(* Logix 5000 project; controller Safety vendor 1 type 14 code 86 rev 19.11; software revision 19.01; part 14 of 17 *)
(* tags used below, declared in another part *)
   FVNR_y778MTR080RC : CONFIGURABLE_ROUT;   // Shear Die Crank Motor FVNR Run Command
   FVR_y702MTR191_Flt : ALIAS FOR Flt_Starter.4;   // Rewind Pinch Roll Starter Fault ( 1= Fault)
   FVR_y702MTR191FC : CONFIGURABLE_ROUT;   // Rewind Pinch Roll FVR Fwd Command
   FVR_y702MTR191RC : CONFIGURABLE_ROUT;   // Rewind Pinch Roll FVR Rev Command
   FVR_y778MTR080_Flt : ALIAS FOR Flt_Starter.5;   // Shear Die Crank Starter Fault ( 1= Fault)
   FVR_y802MTR080_Flt : ALIAS FOR Flt_Starter.6;   // Stacker Side Guide Lift Starter Fault ( 1= Fault)
   FVR_y802MTR080FC : CONFIGURABLE_ROUT;   // Stacker Side Guide Lift FVR Fwd Command
   FVR_y802MTR080RC : CONFIGURABLE_ROUT;   // Stacker Side Guide Lift FVR Rev Command
   FVR_y802MTR230_Flt : ALIAS FOR Flt_Starter.8;   // Scrap Horizontal Conveyor Starter Fault ( 1= Fault)
   FVR_y802MTR230FC : CONFIGURABLE_ROUT;   // Scrap Horizontal Conveyor FVR Fwd Command
   FVR_y802MTR230RC : CONFIGURABLE_ROUT;   // Scrap Horizontal Conveyor FVR Rev Command
   FVR_y802MTR231_Flt : ALIAS FOR Flt_Starter.7;   // Stacker Chain Conveyor Starter Fault ( 1= Fault)
   FVR_y802MTR231FC : CONFIGURABLE_ROUT;   // Stacker Chain Conveyor FVR Fwd Command
   FVR_y802MTR231RC : CONFIGURABLE_ROUT;   // Stacker Chain Conveyor FVR Rev Command
   Line_TotalMode : BOOL;   // Line TOTAL Mode ( 1= Total Mode) (0 = Coil to Coil)
   LineSts : UDT_SysStatus;
   OS11_S1_ModFlt : ALIAS FOR Flt_Modules[1].11;   // OS11 Point I/O Slot01 Module Fault (1 = Fault)
   OS13_S1_ModFlt : ALIAS FOR Flt_Modules[1].12;   // OS13 Point I/O Slot01 Module Fault (1 = Fault)
   OS14_S1_ModFlt : ALIAS FOR Flt_Modules[1].13;   // OS14 Point I/O Slot01 Module Fault (1 = Fault)
   OS15_S1_ModFlt : ALIAS FOR Flt_Modules[1].14;   // OS15 Point I/O Slot01 Module Fault (1 = Fault)
   OS16_S1_ModFlt : ALIAS FOR Flt_Modules[1].15;   // OS16 Point I/O Slot01 Module Fault (1 = Fault)
   OS1_S1_ModFlt : ALIAS FOR Flt_Modules[1].0;   // OS1 Point I/O Slot01 Module Fault (1 = Fault)
   OS2_S1_ModFlt : ALIAS FOR Flt_Modules[1].1;   // OS2 Point I/O Slot01 Module Fault (1 = Fault)
   OS3_S1_ModFlt : ALIAS FOR Flt_Modules[1].2;   // OS3 Point I/O Slot01 Module Fault (1 = Fault)
   OS4N_S1_ModFlt : ALIAS FOR Flt_Modules[1].3;   // OS4N Point I/O Slot01 Module Fault (1 = Fault)
   OS4N_S5_ModFlt : ALIAS FOR Flt_Modules[1].4;   // OS4N Point I/O Slot05 Module Fault (1 = Fault)
   OS4S_S1_ModFlt : ALIAS FOR Flt_Modules[1].5;   // OS4S Point I/O Slot01 Module Fault (1 = Fault)
   OS4S_S5_ModFlt : ALIAS FOR Flt_Modules[1].6;   // OS4S Point I/O Slot05 Module Fault (1 = Fault)
   OS5_S1_ModFlt : ALIAS FOR Flt_Modules[1].7;   // OS5 Point I/O Slot01 Module Fault (1 = Fault)
   OS6_S1_ModFlt : ALIAS FOR Flt_Modules[1].8;   // OS6 Point I/O Slot01 Module Fault (1 = Fault)
   OS8_S1_ModFlt : ALIAS FOR Flt_Modules[1].9;   // OS8 Point I/O Slot01 Module Fault (1 = Fault)
   OS9_S1_ModFlt : ALIAS FOR Flt_Modules[1].10;   // OS9 Point I/O Slot01 Module Fault (1 = Fault)
   RewPR_FVR_En : BOOL;   // Rewind Pinch Roll FVR Enable ( 1= Enable )
   RewPR_FVR_FltRst : BOOL;   // Rewind Pinch Roll Fault Reset ( 1= Reset Cmd )
   RewPR_FVR_FwdCmd : BOOL;   // Rewind Pinch Roll Forward Command ( 1= Run Fwd )
   RewPR_FVR_RevCmd : BOOL;   // Rewind Pinch Roll Reverse Command ( 1= Run Rev)
   ScHorCon_FVR_En : BOOL;   // Scrap Horizontal Conveyor FVR Enable ( 1= Enable )
   ScHorCon_FVR_FltRst : BOOL;   // Scrap Horizontal Conveyor Fault Reset ( 1= Reset Cmd )
   ScHorCon_FVR_FwdCmd : BOOL;   // Scrap Horizontal Conveyor Forward Command ( 1= Run Fwd )
   ScHorCon_FVR_RevCmd : BOOL;   // Scrap Horizontal Conveyor Reverse Command ( 1= Run Rev)
   SftyMap_Mach : DINT[5];   // SAFETY MAPPED From Machine Processor
   SftyMap_ShDie : DINT[5];   // SAFETY MAPPED From Shear Die Processor
   ShearSts : UDT_ShearStatus;
   SkChain_FVR_En : BOOL;   // Stacker Chain FVR Enable ( 1= Enable )
   SkChain_FVR_FltRst : BOOL;   // Stacker Chain Fault Reset ( 1= Reset Cmd )
   SkChain_FVR_FwdCmd : BOOL;   // Stacker Chain Forward Command ( 1= Run Fwd )
   SkChain_FVR_RevCmd : BOOL;   // Stacker Chain Reverse Command ( 1= Run Rev)
   SkSGLift_FVR_En : BOOL;   // Stacker Side Guide Lift FVR Enable ( 1= Enable )
   SkSGLift_FVR_FltRst : BOOL;   // Stacker Side Guide Lift Fault Reset ( 1= Reset Cmd )
   SkSGLift_FVR_FwdCmd : BOOL;   // Stacker Side Guide Lift Forward Command ( 1= Run Fwd )
   SkSGLift_FVR_RevCmd : BOOL;   // Stacker Side Guide Lift Reverse Command ( 1= Run Rev)
   SrDieCrnk_FVNR_En : BOOL;   // Shear Die Crank FVNR Enable ( 1= Enable )
   SrDieCrnk_FVNR_FltRst : BOOL;   // Shear Die Crank FVNR Enable ( 1= Enable )
   SrDieCrnk_FVNR_RunCmd : BOOL;   // Shear Die Crank Run Command ( 1= Run )
   x702MTR191FF : ALIAS FOR MCC1:1:I.Pt00Data;   // Rewind Pinch Roll Fwd Fdbk
   x702MTR191RF : ALIAS FOR MCC1:1:I.Pt01Data;   // Rewind Pinch Roll Rev Fdbk
   x778MTR080RF : ALIAS FOR MCC4:1:I.Pt00Data;   // Shear Crank Motor Run Fdbk
   x802MTR080FF : ALIAS FOR MCC5:1:I.Pt00Data;   // Stacker Side Guide Lift Fwd Fdbk/Up
   x802MTR080RF : ALIAS FOR MCC5:1:I.Pt01Data;   // Stacker Side Guide Lift Rev Fdbk/Down
   x802MTR230FF : ALIAS FOR MCC5:1:I.Pt02Data;   // Scrap Horizontal Conveyor Run Fwd Fdbk
   x802MTR230RF : ALIAS FOR MCC5:1:I.Pt03Data;   // Scrap Horizontal Conveyor Run Rev Fdbk
   x802MTR231FF : ALIAS FOR MCC5:1:I.Pt04Data;   // Stacker Chain Fwd Fdbk
   x802MTR231RF : ALIAS FOR MCC5:1:I.Pt05Data;   // Stacker Chain Rev Fdbk
   y702MTR191FC : ALIAS FOR MCC1:6:O.Pt00Data;   // Rewind Pinch Roll Fwd Cmd
   y702MTR191RC : ALIAS FOR MCC1:6:O.Pt01Data;   // Rewind Pinch Roll Rev Cmd
   y778MTR080RC : ALIAS FOR MCC4:4:O.Pt00Data;   // Shear Die Crank Run Cmd
   y802MTR080FC : ALIAS FOR MCC5:4:O.Pt04Data;   // Stacker Side Guide Lift Fwd Cmd/Up
   y802MTR080RC : ALIAS FOR MCC5:4:O.Pt05Data;   // Stacker Side Guide Lift Rev Cmd/Down
   y802MTR230FC : ALIAS FOR MCC5:4:O.Pt06Data;   // Scrap Horizontal Conveyor Fwd Cmd
   y802MTR230RC : ALIAS FOR MCC5:4:O.Pt07Data;   // Scrap Horizontal Conveyor Rev Cmd
   y802MTR231FC : ALIAS FOR MCC5:5:O.Pt00Data;   // Stacker Chain Fwd Cmd
   y802MTR231RC : ALIAS FOR MCC5:5:O.Pt01Data;   // Stacker Chain Rev Cmd
(* Starters, continued *)

ROUTINE A05_RewPR_FVR   (* ladder *)
// Rewind Pinch Roll
// FVR Starter
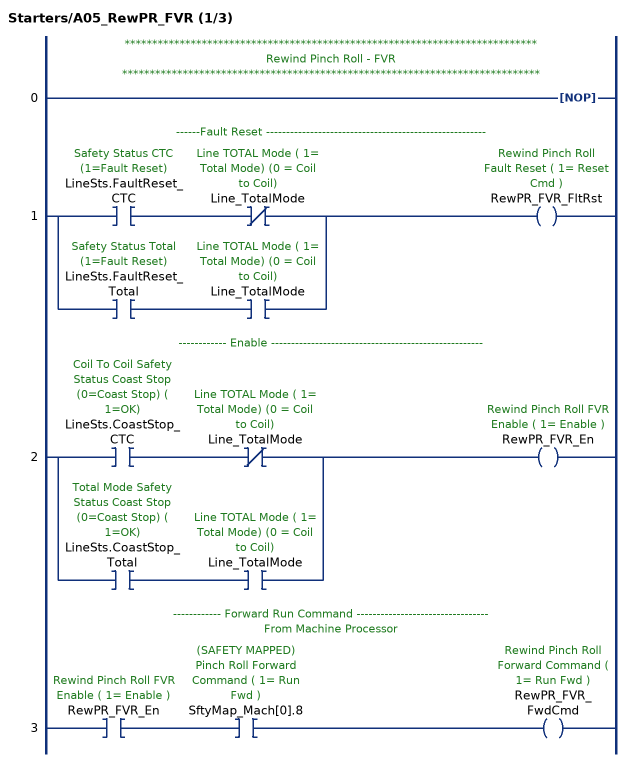
   // ***************************************************************************
   // Rewind Pinch Roll - FVR
   // ****************************************************************************
   0: NOP();
   // ------Fault Reset -------------------------------------------------------
   1: [XIC(LineSts.FaultReset_CTC) XIO(Line_TotalMode) ,XIC(LineSts.FaultReset_Total) XIC(Line_TotalMode) ]OTE(RewPR_FVR_FltRst);
   // ------------ Enable -----------------------------------------------------
   2: [XIC(LineSts.CoastStop_CTC) XIO(Line_TotalMode) ,XIC(LineSts.CoastStop_Total) XIC(Line_TotalMode) ]OTE(RewPR_FVR_En);
   // ------------ Forward Run Command ---------------------------------
   // From Machine Processor
   3: XIC(RewPR_FVR_En)XIC(SftyMap_Mach[0].8)OTE(RewPR_FVR_FwdCmd);
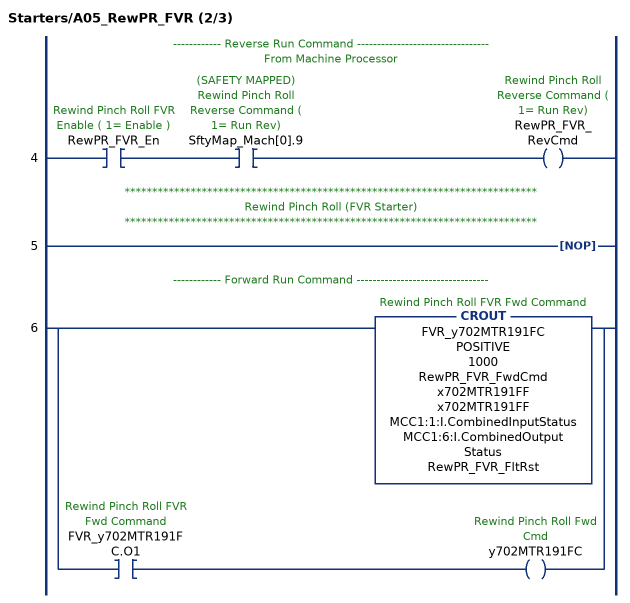
   // ------------ Reverse Run Command ---------------------------------
   // From Machine Processor
   4: XIC(RewPR_FVR_En)XIC(SftyMap_Mach[0].9)OTE(RewPR_FVR_RevCmd);
   // ***************************************************************************
   // Rewind Pinch Roll (FVR Starter)
   // ***************************************************************************
   5: NOP();
   // ------------ Forward Run Command ---------------------------------
   6: [CROUT(FVR_y702MTR191FC,POSITIVE,1000,RewPR_FVR_FwdCmd,x702MTR191FF,x702MTR191FF,MCC1:1:I.CombinedInputStatus,MCC1:6:I.CombinedOutputStatus,RewPR_FVR_FltRst) ,XIC(FVR_y702MTR191FC.O1) OTE(y702MTR191FC) ];
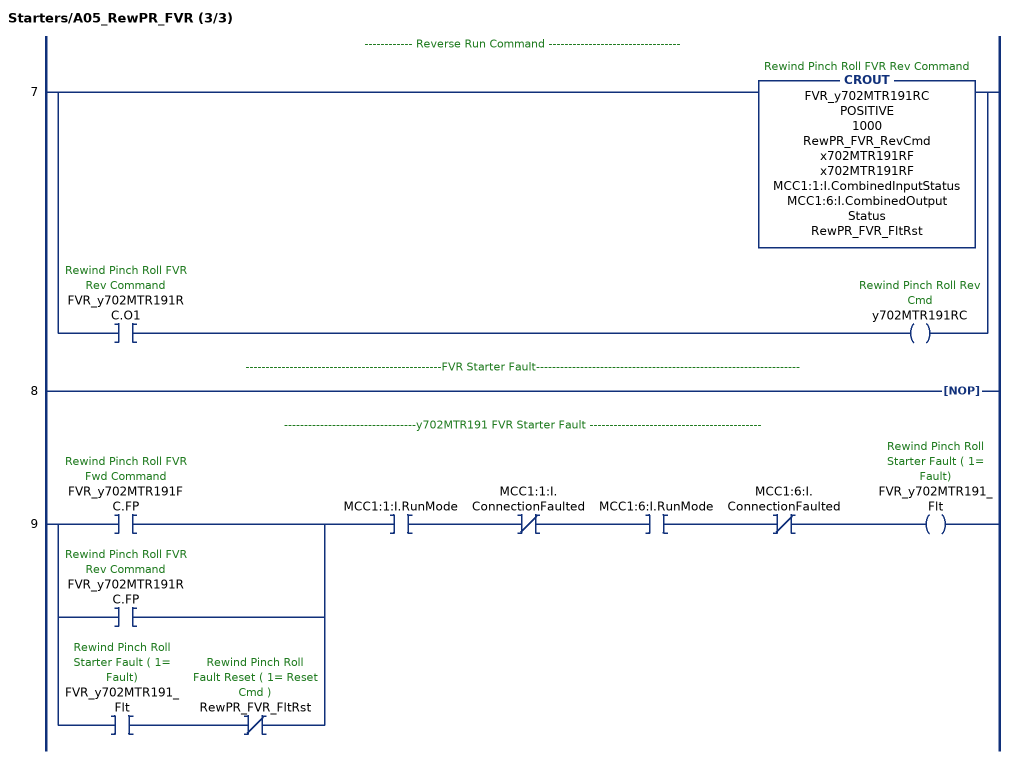
   // ------------ Reverse Run Command ---------------------------------
   7: [CROUT(FVR_y702MTR191RC,POSITIVE,1000,RewPR_FVR_RevCmd,x702MTR191RF,x702MTR191RF,MCC1:1:I.CombinedInputStatus,MCC1:6:I.CombinedOutputStatus,RewPR_FVR_FltRst) ,XIC(FVR_y702MTR191RC.O1) OTE(y702MTR191RC) ];
   // -------------------------------------------------FVR Starter Fault------------------------------------------------------------------
   8: NOP();
   // ---------------------------------y702MTR191 FVR Starter Fault -------------------------------------------
   9: [[XIC(FVR_y702MTR191FC.FP) ,XIC(FVR_y702MTR191RC.FP) ] ,XIC(FVR_y702MTR191_Flt) XIO(RewPR_FVR_FltRst) ]XIC(MCC1:1:I.RunMode)XIO(MCC1:1:I.ConnectionFaulted)XIC(MCC1:6:I.RunMode)XIO(MCC1:6:I.ConnectionFaulted)OTE(FVR_y702MTR191_Flt);
END_ROUTINE

ROUTINE A06_SrDieCrnk_FVNR   (* ladder *)
// Shear Die Crank
// FVNR Starter
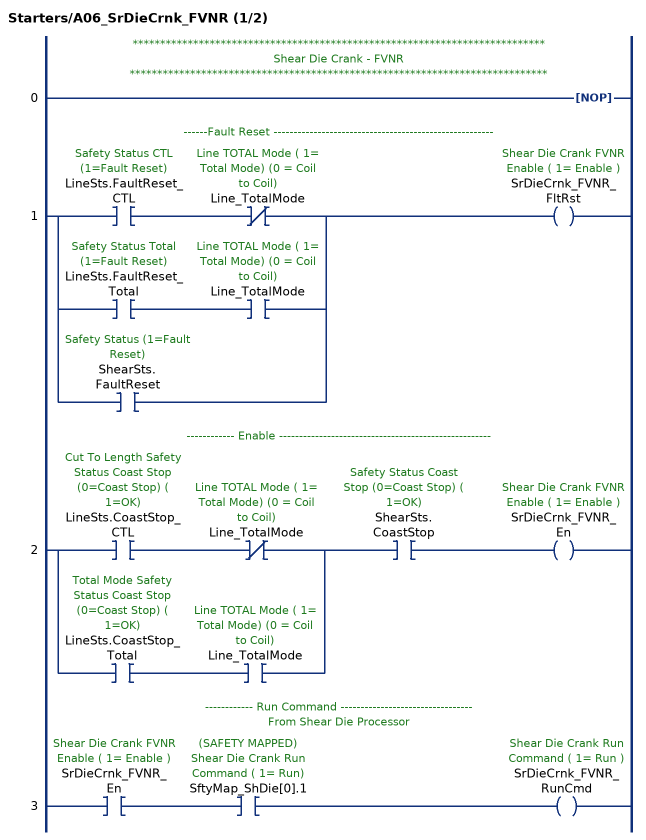
   // ***************************************************************************
   // Shear Die Crank - FVNR
   // ****************************************************************************
   0: NOP();
   // ------Fault Reset -------------------------------------------------------
   1: [XIC(LineSts.FaultReset_CTL) XIO(Line_TotalMode) ,XIC(LineSts.FaultReset_Total) XIC(Line_TotalMode) ,XIC(ShearSts.FaultReset) ]OTE(SrDieCrnk_FVNR_FltRst);
   // ------------ Enable -----------------------------------------------------
   2: [XIC(LineSts.CoastStop_CTL) XIO(Line_TotalMode) ,XIC(LineSts.CoastStop_Total) XIC(Line_TotalMode) ]XIC(ShearSts.CoastStop)OTE(SrDieCrnk_FVNR_En);
   // ------------ Run Command ---------------------------------
   // From Shear Die Processor
   3: XIC(SrDieCrnk_FVNR_En)XIC(SftyMap_ShDie[0].1)OTE(SrDieCrnk_FVNR_RunCmd);
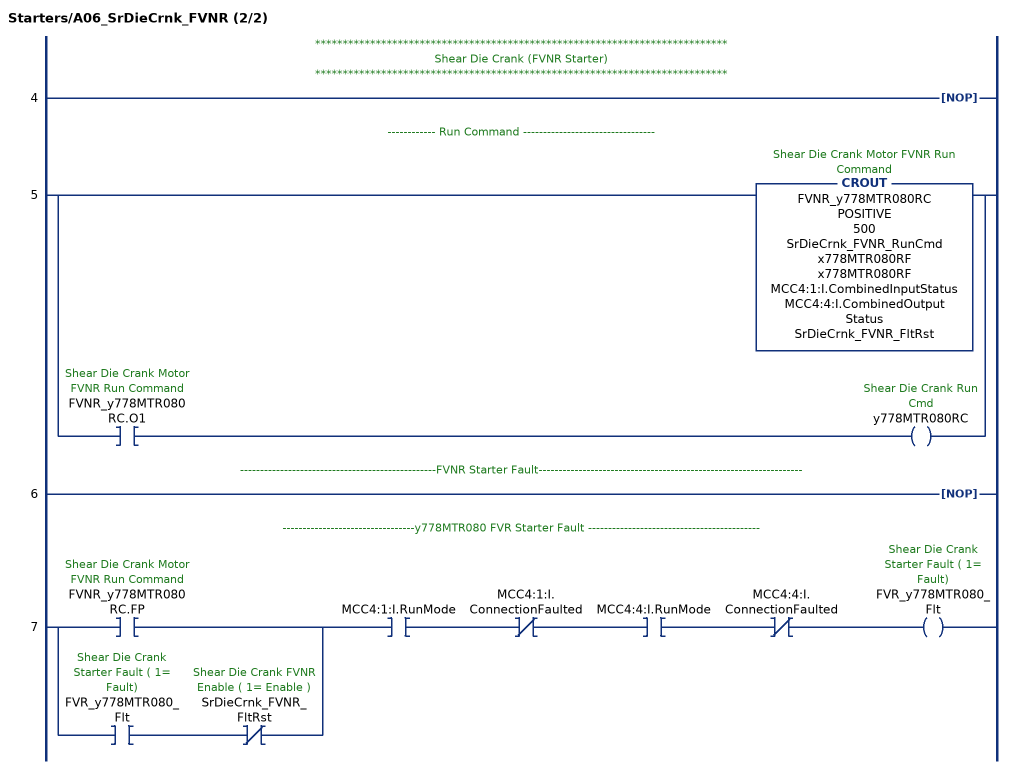
   // ***************************************************************************
   // Shear Die Crank (FVNR Starter)
   // ***************************************************************************
   4: NOP();
   // ------------ Run Command ---------------------------------
   5: [CROUT(FVNR_y778MTR080RC,POSITIVE,500,SrDieCrnk_FVNR_RunCmd,x778MTR080RF,x778MTR080RF,MCC4:1:I.CombinedInputStatus,MCC4:4:I.CombinedOutputStatus,SrDieCrnk_FVNR_FltRst) ,XIC(FVNR_y778MTR080RC.O1) OTE(y778MTR080RC) ];
   // -------------------------------------------------FVNR Starter Fault------------------------------------------------------------------
   6: NOP();
   // ---------------------------------y778MTR080 FVR Starter Fault -------------------------------------------
   7: [XIC(FVNR_y778MTR080RC.FP) ,XIC(FVR_y778MTR080_Flt) XIO(SrDieCrnk_FVNR_FltRst) ]XIC(MCC4:1:I.RunMode)XIO(MCC4:1:I.ConnectionFaulted)XIC(MCC4:4:I.RunMode)XIO(MCC4:4:I.ConnectionFaulted)OTE(FVR_y778MTR080_Flt);
END_ROUTINE

ROUTINE A07_SkSG_FVR   (* ladder *)
// Stacker Side Guide Lift
// FVR Starter
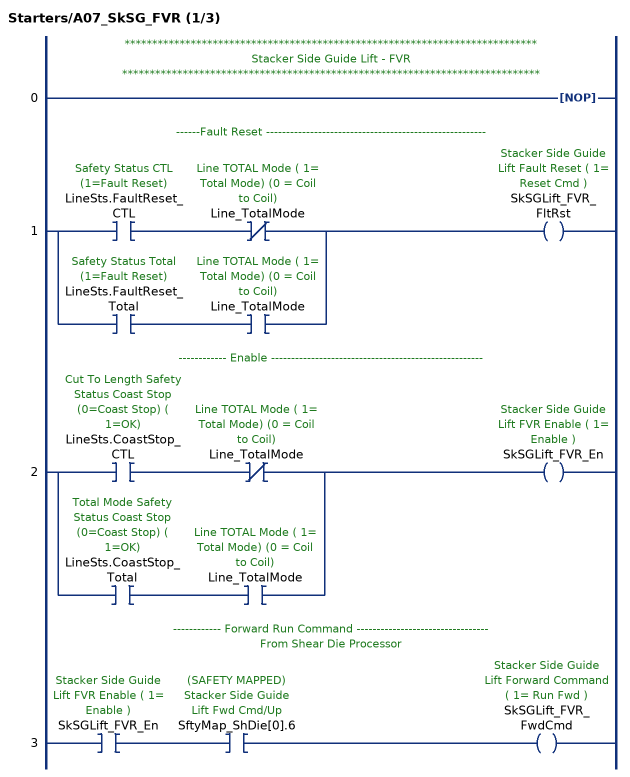
   // ***************************************************************************
   // Stacker Side Guide Lift - FVR
   // ****************************************************************************
   0: NOP();
   // ------Fault Reset -------------------------------------------------------
   1: [XIC(LineSts.FaultReset_CTL) XIO(Line_TotalMode) ,XIC(LineSts.FaultReset_Total) XIC(Line_TotalMode) ]OTE(SkSGLift_FVR_FltRst);
   // ------------ Enable -----------------------------------------------------
   2: [XIC(LineSts.CoastStop_CTL) XIO(Line_TotalMode) ,XIC(LineSts.CoastStop_Total) XIC(Line_TotalMode) ]OTE(SkSGLift_FVR_En);
   // ------------ Forward Run Command ---------------------------------
   // From Shear Die Processor
   3: XIC(SkSGLift_FVR_En)XIC(SftyMap_ShDie[0].6)OTE(SkSGLift_FVR_FwdCmd);
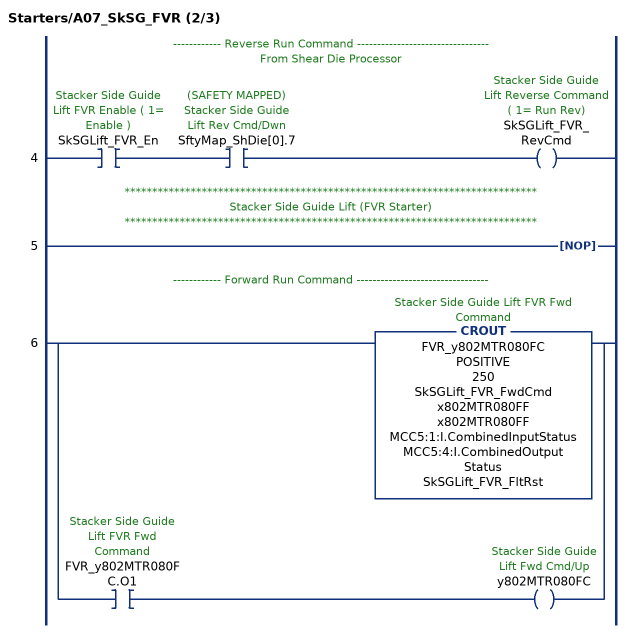
   // ------------ Reverse Run Command ---------------------------------
   // From Shear Die Processor
   4: XIC(SkSGLift_FVR_En)XIC(SftyMap_ShDie[0].7)OTE(SkSGLift_FVR_RevCmd);
   // ***************************************************************************
   // Stacker Side Guide Lift (FVR Starter)
   // ***************************************************************************
   5: NOP();
   // ------------ Forward Run Command ---------------------------------
   6: [CROUT(FVR_y802MTR080FC,POSITIVE,250,SkSGLift_FVR_FwdCmd,x802MTR080FF,x802MTR080FF,MCC5:1:I.CombinedInputStatus,MCC5:4:I.CombinedOutputStatus,SkSGLift_FVR_FltRst) ,XIC(FVR_y802MTR080FC.O1) OTE(y802MTR080FC) ];
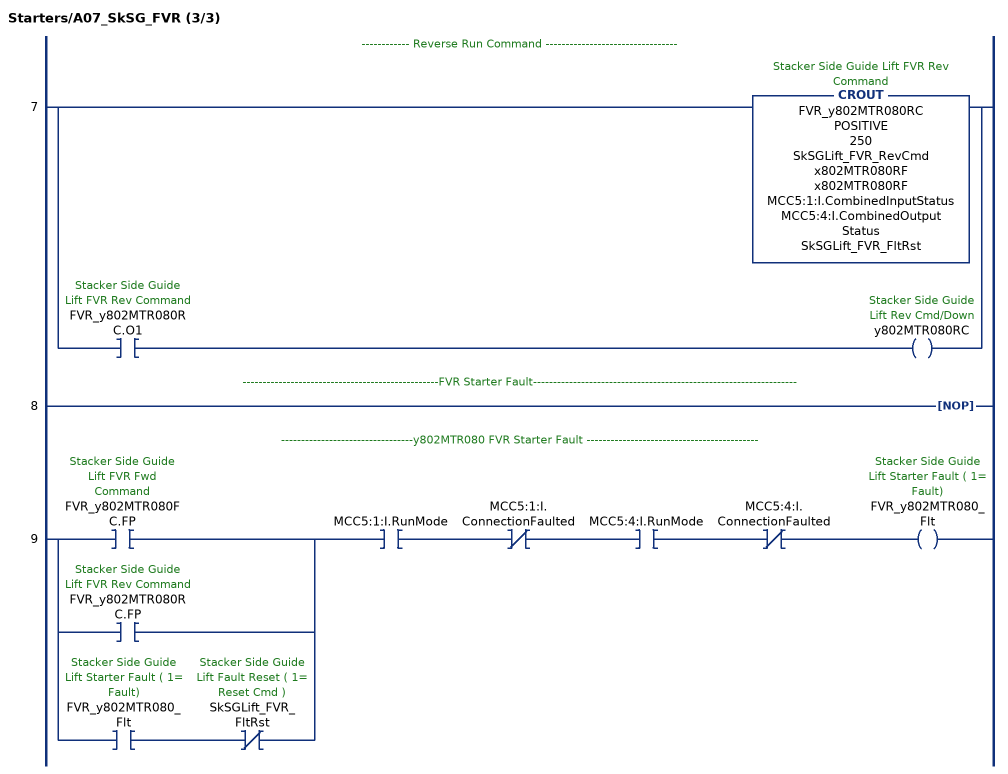
   // ------------ Reverse Run Command ---------------------------------
   7: [CROUT(FVR_y802MTR080RC,POSITIVE,250,SkSGLift_FVR_RevCmd,x802MTR080RF,x802MTR080RF,MCC5:1:I.CombinedInputStatus,MCC5:4:I.CombinedOutputStatus,SkSGLift_FVR_FltRst) ,XIC(FVR_y802MTR080RC.O1) OTE(y802MTR080RC) ];
   // -------------------------------------------------FVR Starter Fault------------------------------------------------------------------
   8: NOP();
   // ---------------------------------y802MTR080 FVR Starter Fault -------------------------------------------
   9: [[XIC(FVR_y802MTR080FC.FP) ,XIC(FVR_y802MTR080RC.FP) ] ,XIC(FVR_y802MTR080_Flt) XIO(SkSGLift_FVR_FltRst) ]XIC(MCC5:1:I.RunMode)XIO(MCC5:1:I.ConnectionFaulted)XIC(MCC5:4:I.RunMode)XIO(MCC5:4:I.ConnectionFaulted)OTE(FVR_y802MTR080_Flt);
END_ROUTINE

ROUTINE A08_SkChain_FVR   (* ladder *)
// Stacker Chain Conveyor
// FVR Starter
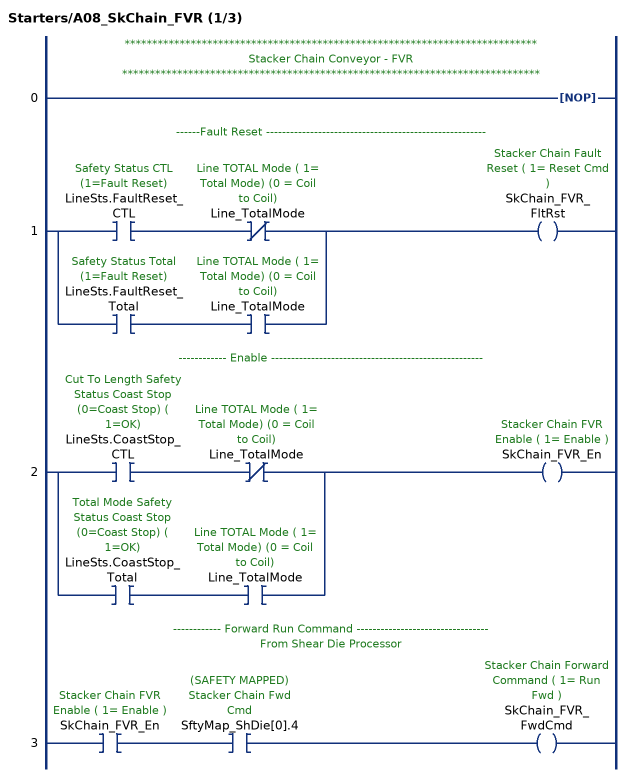
   // ***************************************************************************
   // Stacker Chain Conveyor - FVR
   // ****************************************************************************
   0: NOP();
   // ------Fault Reset -------------------------------------------------------
   1: [XIC(LineSts.FaultReset_CTL) XIO(Line_TotalMode) ,XIC(LineSts.FaultReset_Total) XIC(Line_TotalMode) ]OTE(SkChain_FVR_FltRst);
   // ------------ Enable -----------------------------------------------------
   2: [XIC(LineSts.CoastStop_CTL) XIO(Line_TotalMode) ,XIC(LineSts.CoastStop_Total) XIC(Line_TotalMode) ]OTE(SkChain_FVR_En);
   // ------------ Forward Run Command ---------------------------------
   // From Shear Die Processor
   3: XIC(SkChain_FVR_En)XIC(SftyMap_ShDie[0].4)OTE(SkChain_FVR_FwdCmd);
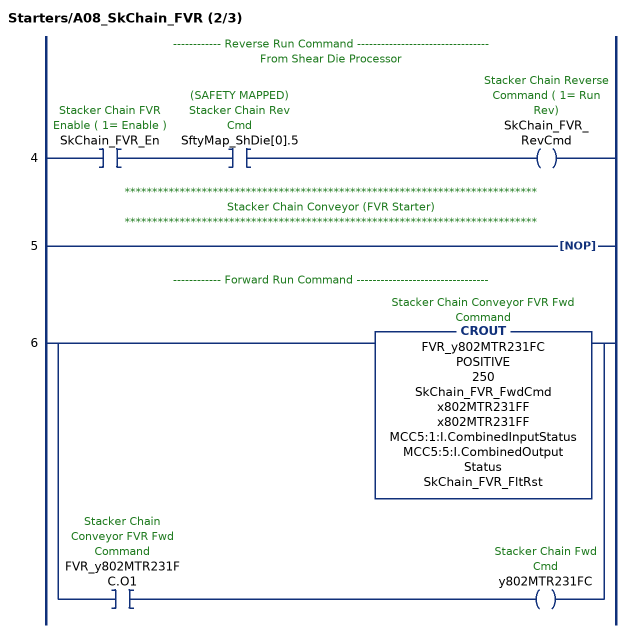
   // ------------ Reverse Run Command ---------------------------------
   // From Shear Die Processor
   4: XIC(SkChain_FVR_En)XIC(SftyMap_ShDie[0].5)OTE(SkChain_FVR_RevCmd);
   // ***************************************************************************
   // Stacker Chain Conveyor (FVR Starter)
   // ***************************************************************************
   5: NOP();
   // ------------ Forward Run Command ---------------------------------
   6: [CROUT(FVR_y802MTR231FC,POSITIVE,250,SkChain_FVR_FwdCmd,x802MTR231FF,x802MTR231FF,MCC5:1:I.CombinedInputStatus,MCC5:5:I.CombinedOutputStatus,SkChain_FVR_FltRst) ,XIC(FVR_y802MTR231FC.O1) OTE(y802MTR231FC) ];
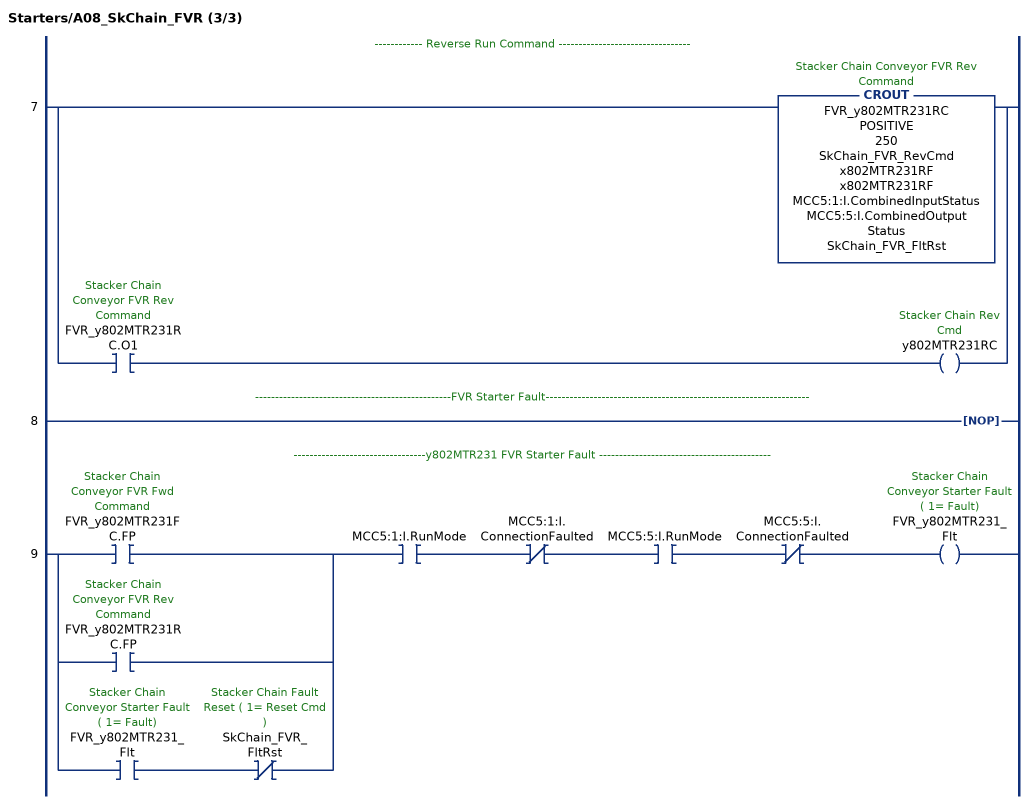
   // ------------ Reverse Run Command ---------------------------------
   7: [CROUT(FVR_y802MTR231RC,POSITIVE,250,SkChain_FVR_RevCmd,x802MTR231RF,x802MTR231RF,MCC5:1:I.CombinedInputStatus,MCC5:5:I.CombinedOutputStatus,SkChain_FVR_FltRst) ,XIC(FVR_y802MTR231RC.O1) OTE(y802MTR231RC) ];
   // -------------------------------------------------FVR Starter Fault------------------------------------------------------------------
   8: NOP();
   // ---------------------------------y802MTR231 FVR Starter Fault -------------------------------------------
   9: [[XIC(FVR_y802MTR231FC.FP) ,XIC(FVR_y802MTR231RC.FP) ] ,XIC(FVR_y802MTR231_Flt) XIO(SkChain_FVR_FltRst) ]XIC(MCC5:1:I.RunMode)XIO(MCC5:1:I.ConnectionFaulted)XIC(MCC5:5:I.RunMode)XIO(MCC5:5:I.ConnectionFaulted)OTE(FVR_y802MTR231_Flt);
END_ROUTINE

ROUTINE A09_ScHorCon_FVR   (* ladder *)
// Scrap Horizontal Conveyor
// FVR Starter
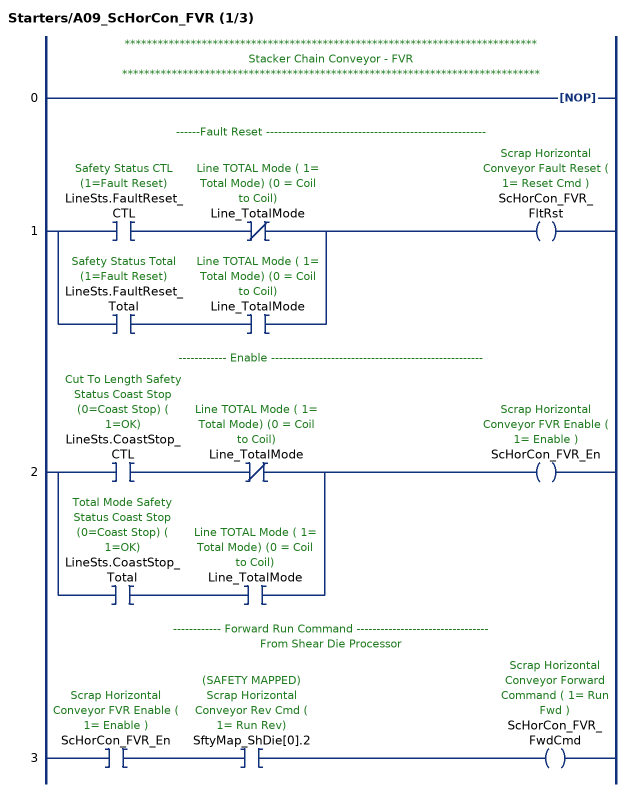
   // ***************************************************************************
   // Stacker Chain Conveyor - FVR
   // ****************************************************************************
   0: NOP();
   // ------Fault Reset -------------------------------------------------------
   1: [XIC(LineSts.FaultReset_CTL) XIO(Line_TotalMode) ,XIC(LineSts.FaultReset_Total) XIC(Line_TotalMode) ]OTE(ScHorCon_FVR_FltRst);
   // ------------ Enable -----------------------------------------------------
   2: [XIC(LineSts.CoastStop_CTL) XIO(Line_TotalMode) ,XIC(LineSts.CoastStop_Total) XIC(Line_TotalMode) ]OTE(ScHorCon_FVR_En);
   // ------------ Forward Run Command ---------------------------------
   // From Shear Die Processor
   3: XIC(ScHorCon_FVR_En)XIC(SftyMap_ShDie[0].2)OTE(ScHorCon_FVR_FwdCmd);
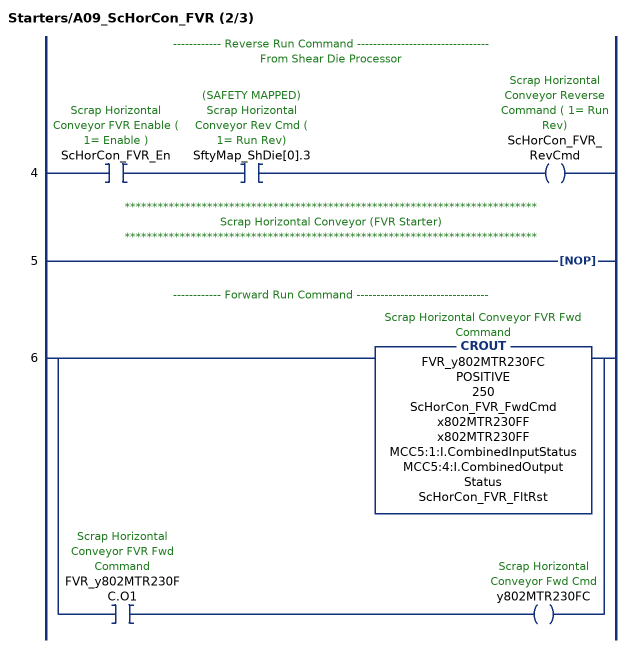
   // ------------ Reverse Run Command ---------------------------------
   // From Shear Die Processor
   4: XIC(ScHorCon_FVR_En)XIC(SftyMap_ShDie[0].3)OTE(ScHorCon_FVR_RevCmd);
   // ***************************************************************************
   // Scrap Horizontal Conveyor (FVR Starter)
   // ***************************************************************************
   5: NOP();
   // ------------ Forward Run Command ---------------------------------
   6: [CROUT(FVR_y802MTR230FC,POSITIVE,250,ScHorCon_FVR_FwdCmd,x802MTR230FF,x802MTR230FF,MCC5:1:I.CombinedInputStatus,MCC5:4:I.CombinedOutputStatus,ScHorCon_FVR_FltRst) ,XIC(FVR_y802MTR230FC.O1) OTE(y802MTR230FC) ];
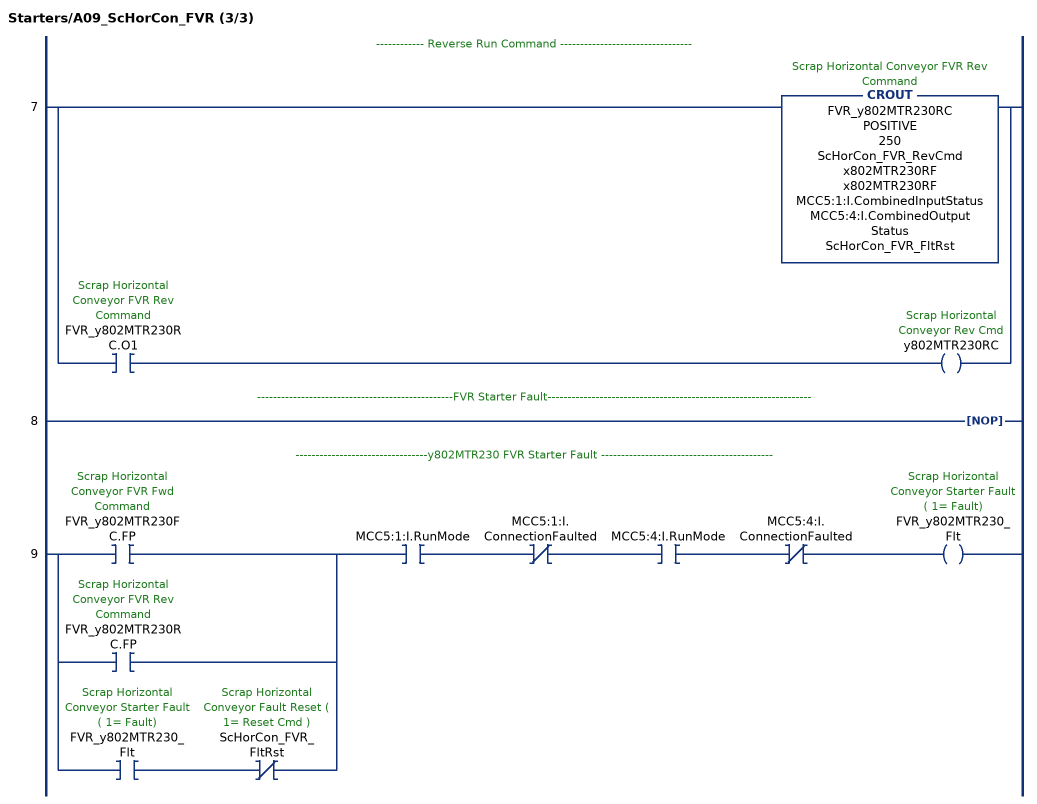
   // ------------ Reverse Run Command ---------------------------------
   7: [CROUT(FVR_y802MTR230RC,POSITIVE,250,ScHorCon_FVR_RevCmd,x802MTR230RF,x802MTR230RF,MCC5:1:I.CombinedInputStatus,MCC5:4:I.CombinedOutputStatus,ScHorCon_FVR_FltRst) ,XIC(FVR_y802MTR230RC.O1) OTE(y802MTR230RC) ];
   // -------------------------------------------------FVR Starter Fault------------------------------------------------------------------
   8: NOP();
   // ---------------------------------y802MTR230 FVR Starter Fault -------------------------------------------
   9: [[XIC(FVR_y802MTR230FC.FP) ,XIC(FVR_y802MTR230RC.FP) ] ,XIC(FVR_y802MTR230_Flt) XIO(ScHorCon_FVR_FltRst) ]XIC(MCC5:1:I.RunMode)XIO(MCC5:1:I.ConnectionFaulted)XIC(MCC5:4:I.RunMode)XIO(MCC5:4:I.ConnectionFaulted)OTE(FVR_y802MTR230_Flt);
END_ROUTINE
END_PROGRAM

PROGRAM System   (* main routine MainRoutine *)
// Safety System Logic

ROUTINE A01_SftyModFlts_OS   (* ladder *)
// Operator Station
// Safety Module Faults
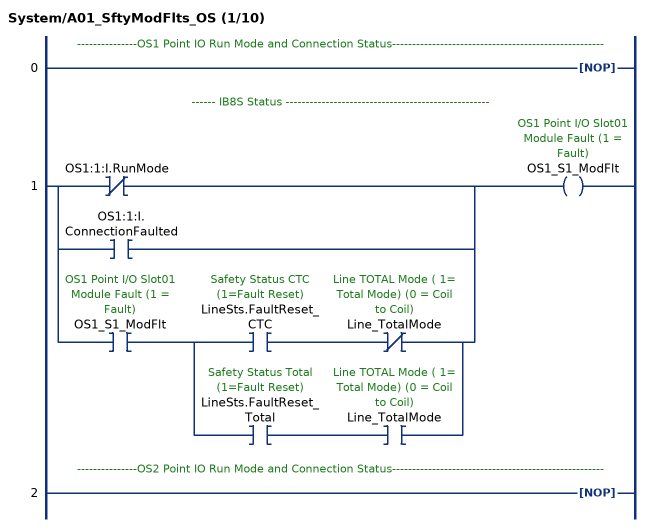
   // ---------------OS1 Point IO Run Mode and Connection Status-----------------------------------------------------
   0: NOP();
   // ------ IB8S Status ---------------------------------------------------
   1: [XIO(OS1:1:I.RunMode) ,XIC(OS1:1:I.ConnectionFaulted) ,XIC(OS1_S1_ModFlt) [XIC(LineSts.FaultReset_CTC) XIO(Line_TotalMode) ,XIC(LineSts.FaultReset_Total) XIC(Line_TotalMode) ] ]OTE(OS1_S1_ModFlt);
   // ---------------OS2 Point IO Run Mode and Connection Status-----------------------------------------------------
   2: NOP();
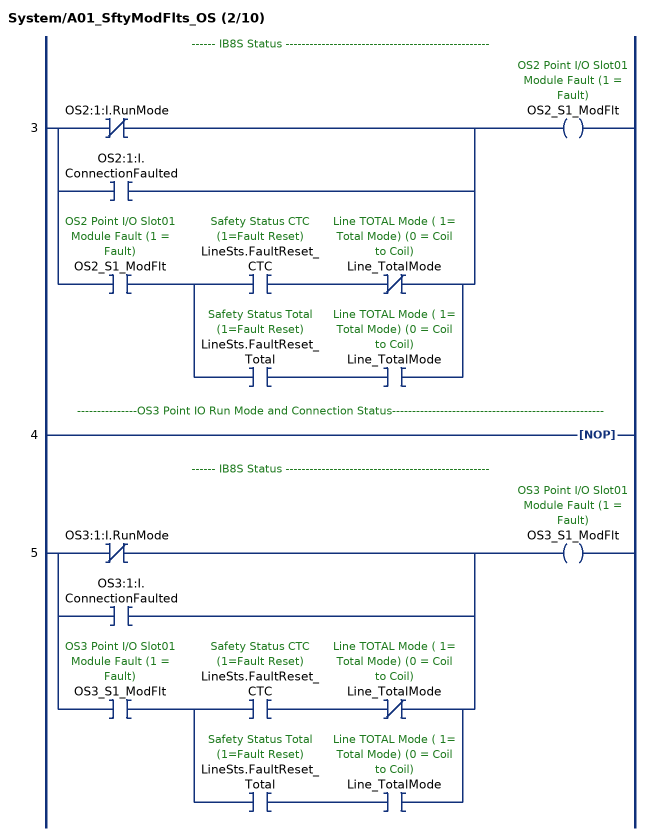
   // ------ IB8S Status ---------------------------------------------------
   3: [XIO(OS2:1:I.RunMode) ,XIC(OS2:1:I.ConnectionFaulted) ,XIC(OS2_S1_ModFlt) [XIC(LineSts.FaultReset_CTC) XIO(Line_TotalMode) ,XIC(LineSts.FaultReset_Total) XIC(Line_TotalMode) ] ]OTE(OS2_S1_ModFlt);
   // ---------------OS3 Point IO Run Mode and Connection Status-----------------------------------------------------
   4: NOP();
   // ------ IB8S Status ---------------------------------------------------
   5: [XIO(OS3:1:I.RunMode) ,XIC(OS3:1:I.ConnectionFaulted) ,XIC(OS3_S1_ModFlt) [XIC(LineSts.FaultReset_CTC) XIO(Line_TotalMode) ,XIC(LineSts.FaultReset_Total) XIC(Line_TotalMode) ] ]OTE(OS3_S1_ModFlt);
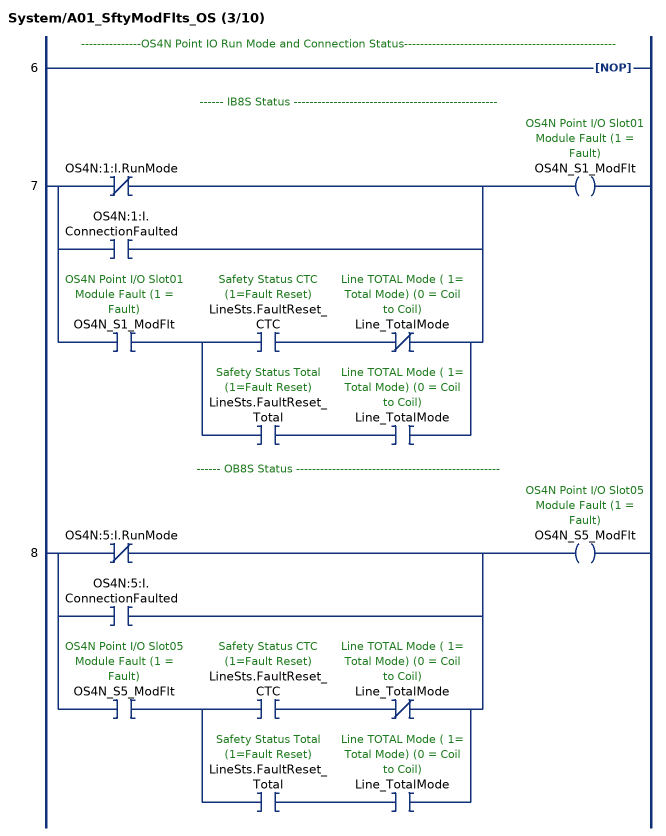
   // ---------------OS4N Point IO Run Mode and Connection Status-----------------------------------------------------
   6: NOP();
   // ------ IB8S Status ---------------------------------------------------
   7: [XIO(OS4N:1:I.RunMode) ,XIC(OS4N:1:I.ConnectionFaulted) ,XIC(OS4N_S1_ModFlt) [XIC(LineSts.FaultReset_CTC) XIO(Line_TotalMode) ,XIC(LineSts.FaultReset_Total) XIC(Line_TotalMode) ] ]OTE(OS4N_S1_ModFlt);
   // ------ OB8S Status ---------------------------------------------------
   8: [XIO(OS4N:5:I.RunMode) ,XIC(OS4N:5:I.ConnectionFaulted) ,XIC(OS4N_S5_ModFlt) [XIC(LineSts.FaultReset_CTC) XIO(Line_TotalMode) ,XIC(LineSts.FaultReset_Total) XIC(Line_TotalMode) ] ]OTE(OS4N_S5_ModFlt);
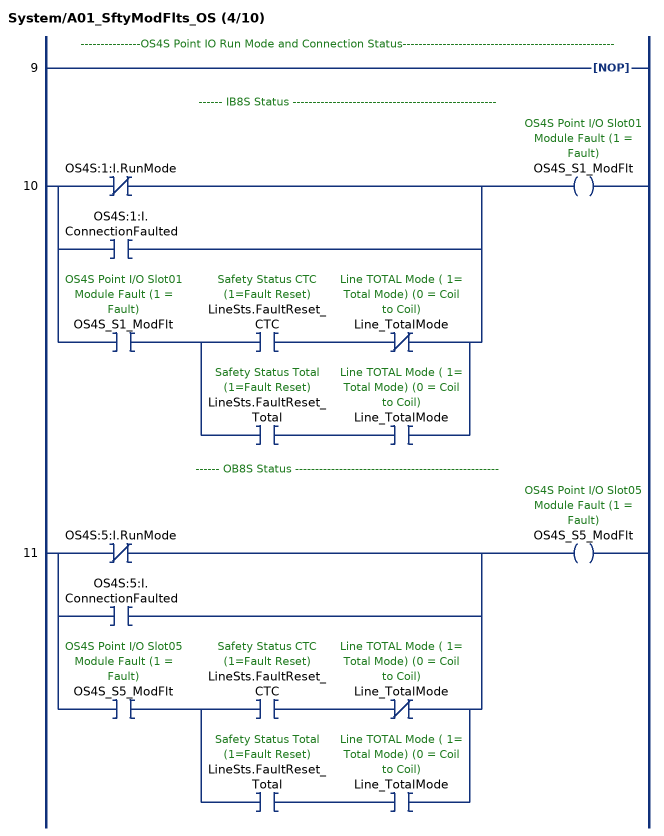
   // ---------------OS4S Point IO Run Mode and Connection Status-----------------------------------------------------
   9: NOP();
   // ------ IB8S Status ---------------------------------------------------
   10: [XIO(OS4S:1:I.RunMode) ,XIC(OS4S:1:I.ConnectionFaulted) ,XIC(OS4S_S1_ModFlt) [XIC(LineSts.FaultReset_CTC) XIO(Line_TotalMode) ,XIC(LineSts.FaultReset_Total) XIC(Line_TotalMode) ] ]OTE(OS4S_S1_ModFlt);
   // ------ OB8S Status ---------------------------------------------------
   11: [XIO(OS4S:5:I.RunMode) ,XIC(OS4S:5:I.ConnectionFaulted) ,XIC(OS4S_S5_ModFlt) [XIC(LineSts.FaultReset_CTC) XIO(Line_TotalMode) ,XIC(LineSts.FaultReset_Total) XIC(Line_TotalMode) ] ]OTE(OS4S_S5_ModFlt);
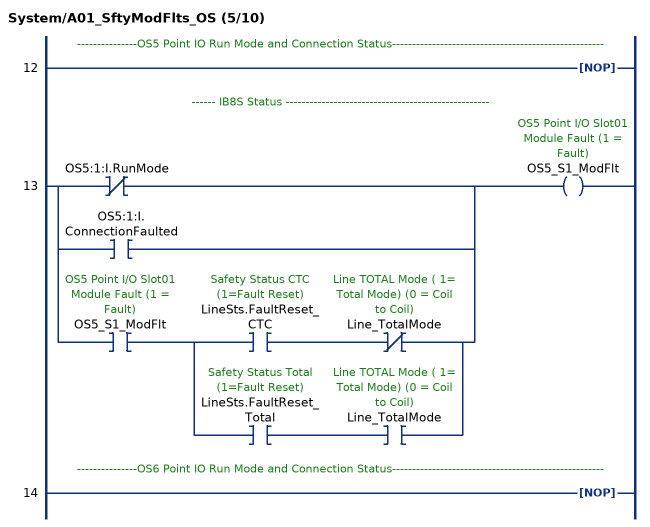
   // ---------------OS5 Point IO Run Mode and Connection Status-----------------------------------------------------
   12: NOP();
   // ------ IB8S Status ---------------------------------------------------
   13: [XIO(OS5:1:I.RunMode) ,XIC(OS5:1:I.ConnectionFaulted) ,XIC(OS5_S1_ModFlt) [XIC(LineSts.FaultReset_CTC) XIO(Line_TotalMode) ,XIC(LineSts.FaultReset_Total) XIC(Line_TotalMode) ] ]OTE(OS5_S1_ModFlt);
   // ---------------OS6 Point IO Run Mode and Connection Status-----------------------------------------------------
   14: NOP();
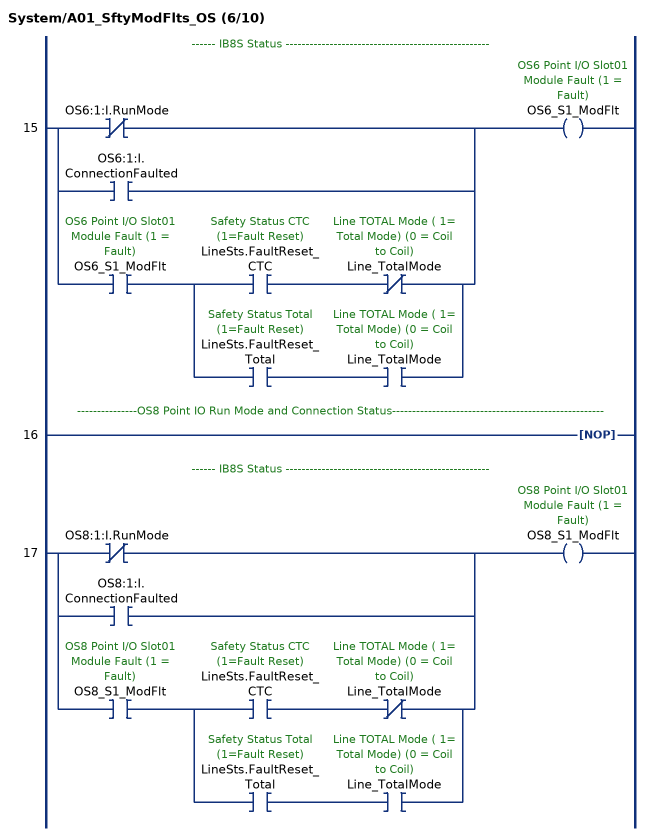
   // ------ IB8S Status ---------------------------------------------------
   15: [XIO(OS6:1:I.RunMode) ,XIC(OS6:1:I.ConnectionFaulted) ,XIC(OS6_S1_ModFlt) [XIC(LineSts.FaultReset_CTC) XIO(Line_TotalMode) ,XIC(LineSts.FaultReset_Total) XIC(Line_TotalMode) ] ]OTE(OS6_S1_ModFlt);
   // ---------------OS8 Point IO Run Mode and Connection Status-----------------------------------------------------
   16: NOP();
   // ------ IB8S Status ---------------------------------------------------
   17: [XIO(OS8:1:I.RunMode) ,XIC(OS8:1:I.ConnectionFaulted) ,XIC(OS8_S1_ModFlt) [XIC(LineSts.FaultReset_CTC) XIO(Line_TotalMode) ,XIC(LineSts.FaultReset_Total) XIC(Line_TotalMode) ] ]OTE(OS8_S1_ModFlt);
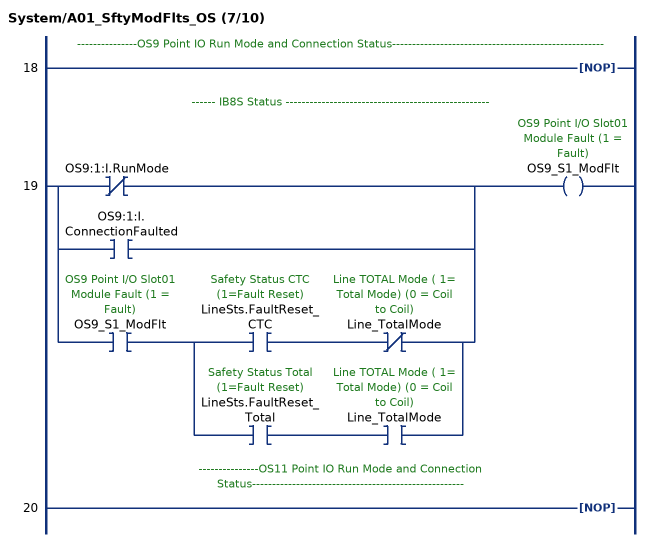
   // ---------------OS9 Point IO Run Mode and Connection Status-----------------------------------------------------
   18: NOP();
   // ------ IB8S Status ---------------------------------------------------
   19: [XIO(OS9:1:I.RunMode) ,XIC(OS9:1:I.ConnectionFaulted) ,XIC(OS9_S1_ModFlt) [XIC(LineSts.FaultReset_CTC) XIO(Line_TotalMode) ,XIC(LineSts.FaultReset_Total) XIC(Line_TotalMode) ] ]OTE(OS9_S1_ModFlt);
   // ---------------OS11 Point IO Run Mode and Connection Status-----------------------------------------------------
   20: NOP();
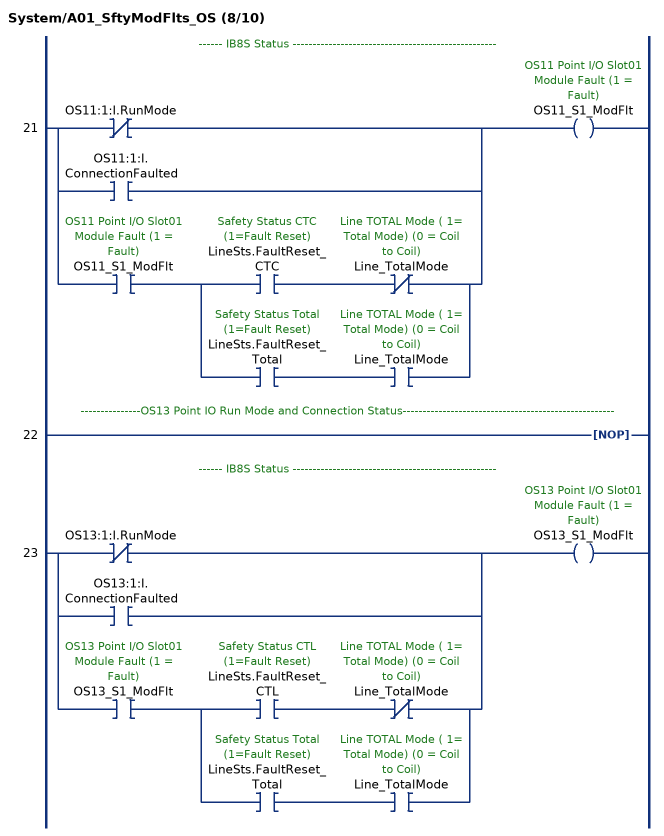
   // ------ IB8S Status ---------------------------------------------------
   21: [XIO(OS11:1:I.RunMode) ,XIC(OS11:1:I.ConnectionFaulted) ,XIC(OS11_S1_ModFlt) [XIC(LineSts.FaultReset_CTC) XIO(Line_TotalMode) ,XIC(LineSts.FaultReset_Total) XIC(Line_TotalMode) ] ]OTE(OS11_S1_ModFlt);
   // ---------------OS13 Point IO Run Mode and Connection Status-----------------------------------------------------
   22: NOP();
   // ------ IB8S Status ---------------------------------------------------
   23: [XIO(OS13:1:I.RunMode) ,XIC(OS13:1:I.ConnectionFaulted) ,XIC(OS13_S1_ModFlt) [XIC(LineSts.FaultReset_CTL) XIO(Line_TotalMode) ,XIC(LineSts.FaultReset_Total) XIC(Line_TotalMode) ] ]OTE(OS13_S1_ModFlt);
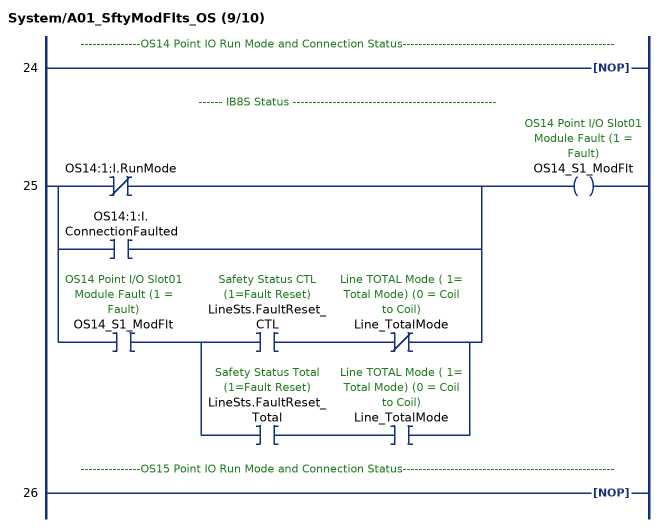
   // ---------------OS14 Point IO Run Mode and Connection Status-----------------------------------------------------
   24: NOP();
   // ------ IB8S Status ---------------------------------------------------
   25: [XIO(OS14:1:I.RunMode) ,XIC(OS14:1:I.ConnectionFaulted) ,XIC(OS14_S1_ModFlt) [XIC(LineSts.FaultReset_CTL) XIO(Line_TotalMode) ,XIC(LineSts.FaultReset_Total) XIC(Line_TotalMode) ] ]OTE(OS14_S1_ModFlt);
   // ---------------OS15 Point IO Run Mode and Connection Status-----------------------------------------------------
   26: NOP();
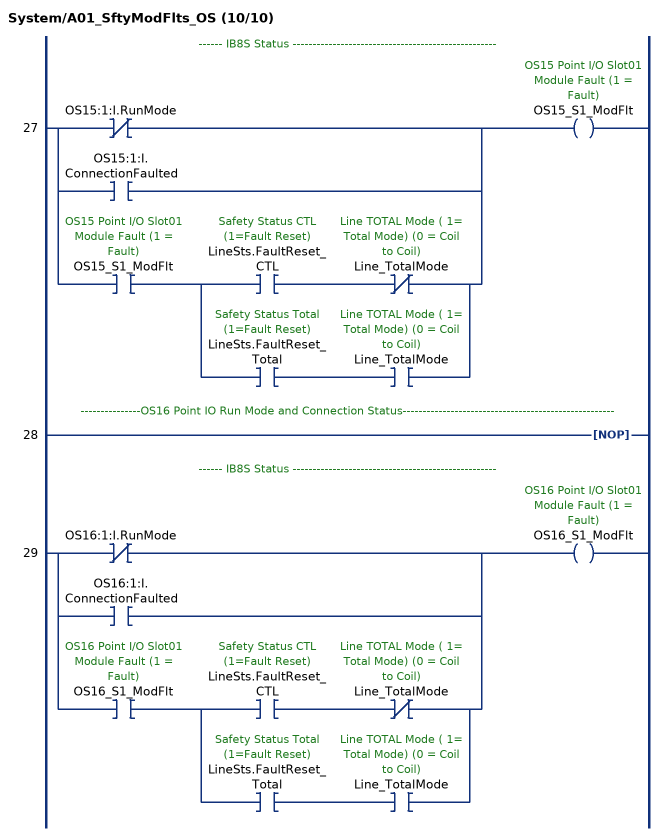
   // ------ IB8S Status ---------------------------------------------------
   27: [XIO(OS15:1:I.RunMode) ,XIC(OS15:1:I.ConnectionFaulted) ,XIC(OS15_S1_ModFlt) [XIC(LineSts.FaultReset_CTL) XIO(Line_TotalMode) ,XIC(LineSts.FaultReset_Total) XIC(Line_TotalMode) ] ]OTE(OS15_S1_ModFlt);
   // ---------------OS16 Point IO Run Mode and Connection Status-----------------------------------------------------
   28: NOP();
   // ------ IB8S Status ---------------------------------------------------
   29: [XIO(OS16:1:I.RunMode) ,XIC(OS16:1:I.ConnectionFaulted) ,XIC(OS16_S1_ModFlt) [XIC(LineSts.FaultReset_CTL) XIO(Line_TotalMode) ,XIC(LineSts.FaultReset_Total) XIC(Line_TotalMode) ] ]OTE(OS16_S1_ModFlt);
END_ROUTINE
